FUNCTION_BLOCK FB_Coordinador_SFC
VAR_IN_OUT

	UnidadesPendientes: UINT;
	UnidadesRealizadas: UINT;

END_VAR
VAR_INPUT

	//  SFC-Flags
	SFCPause: BOOL;
	SFCReset: BOOL;
	
	// Indicadores de sincronización
	Ack: BOOL:= TRUE;
	Execute: BOOL;
	
	// Parámetros de sincronización
	BaseSituada: BOOL;
	PaleSituado: BOOL;
	PaleVerificado: BOOL;
	PaleDesechado: BOOL;
	PaleTransferido: BOOL;
	BaseTransferida: BOOL;
	
	// Parámetros
	CondicionInicial: BOOL;
	UnidadesSolicitadas: UINT;	

END_VAR
VAR_OUTPUT
	
	// Indicadores de sincronización
	Done: BOOL;
	Ready: BOOL;
	
	// Parámetros de sincronización
	SituaBase: BOOL;
	SituaPale: BOOL;
	VerificaPale: BOOL;
	DesechaPale: BOOL;
	TransfierePale: BOOL;
	TransfiereBase: BOOL;
	
	// Salidas
	LamparaAlarma: BOOL;
	LamparaMarcha: BOOL;
	
END_VAR
VAR
	
	// Bloques funcionales	
	CLK: FB_Clock;
	
END_VAR

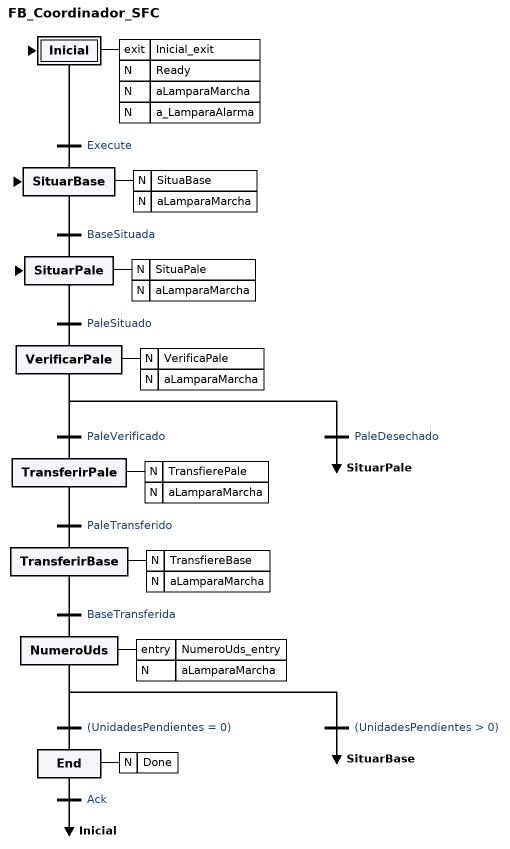
INITIAL_STEP Inicial:
    Inicial_exit(P0);  // exit action
    Ready(N);
    aLamparaMarcha(N);
    a_LamparaAlarma(N);
END_STEP
TRANSITION FROM Inicial TO SituarBase
    := Execute;
END_TRANSITION
STEP SituarBase:
    SituaBase(N);
    aLamparaMarcha(N);
END_STEP
TRANSITION FROM SituarBase TO SituarPale
    := BaseSituada;
END_TRANSITION
STEP SituarPale:
    SituaPale(N);
    aLamparaMarcha(N);
END_STEP
TRANSITION FROM SituarPale TO VerificarPale
    := PaleSituado;
END_TRANSITION
STEP VerificarPale:
    VerificaPale(N);
    aLamparaMarcha(N);
END_STEP
TRANSITION FROM VerificarPale TO TransferirPale
    := PaleVerificado;
END_TRANSITION
STEP TransferirPale:
    TransfierePale(N);
    aLamparaMarcha(N);
END_STEP
TRANSITION FROM TransferirPale TO TransferirBase
    := PaleTransferido;
END_TRANSITION
STEP TransferirBase:
    TransfiereBase(N);
    aLamparaMarcha(N);
END_STEP
TRANSITION FROM TransferirBase TO NumeroUds
    := BaseTransferida;
END_TRANSITION
STEP NumeroUds:
    NumeroUds_entry(P1);  // entry action
    aLamparaMarcha(N);
END_STEP
TRANSITION FROM NumeroUds TO End
    := (UnidadesPendientes = 0);
END_TRANSITION
TRANSITION FROM NumeroUds TO SituarBase
    := (UnidadesPendientes > 0);
END_TRANSITION
STEP End:
    Done(N);
END_STEP
TRANSITION FROM End TO Inicial
    := Ack;
END_TRANSITION
TRANSITION FROM VerificarPale TO SituarPale
    := PaleDesechado;
END_TRANSITION

ACTION a_LamparaAlarma:
LamparaAlarma := (Inicial.x AND NOT CondicionInicial AND CLK.Q);
END_ACTION

ACTION aLamparaMarcha:
LamparaMarcha := (Inicial.x AND NOT CondicionInicial AND CLK.Q) OR NOT Inicial.x;
END_ACTION

ACTION Inicial_exit:
// Al iniciar una tarea se actualiza las unidades pendientes
IF (UnidadesPendientes = 0) THEN
    UnidadesPendientes := UnidadesSolicitadas;
END_IF
END_ACTION

ACTION NumeroUds_entry:
// Al completar una transferencia actualizamos los valores de los contadores
UnidadesRealizadas := UnidadesRealizadas + 1;

IF (UnidadesPendientes > 0) THEN
	UnidadesPendientes := UnidadesPendientes - 1;
END_IF
END_ACTION

END_FUNCTION_BLOCK

(* stored: Version 1.1.0.1, ProductVersion 3.1.4024.12
   POU FB_Coordinador_SFC: Id {39e99b26-ca1b-4e0c-9027-108f648dd0e2}, SpecialFunc None
   Action a_LamparaAlarma: Id {59612ca8-7fe3-47f0-a41f-70c4610b3503}
   Action aLamparaMarcha: Id {5f208487-2a26-447e-a98a-cdcb80d410a6}
   Action Inicial_exit: Id {943ebe45-7cb7-4429-86bb-557c2de4fe51}
   Action NumeroUds_entry: Id {1a8f7e27-62e1-4e59-a16c-778c45ece5ea} *)
